// TIA Portal V17 export
// export: Created 2023-05-07T12:12:11.3887996Z, ExportSetting WithDefaults, DisplayName Totally Integrated Automation Portal, DisplayVersion V17, DisplayName TIA Portal Openness, DisplayVersion V17, DisplayName TIA Portal Version Control Interface, DisplayVersion V17, DisplayName TIA Portal Test Suite Advanced, DisplayVersion V17, DisplayName STEP 7 Professional, DisplayVersion V17, DisplayName SIMATIC Energy Suite, DisplayVersion V17, DisplayName STEP 7 Safety, DisplayVersion V17, DisplayName WinCC Professional, DisplayVersion V17
FUNCTION "TrainingFunction" : Void   // FC7, LAD
TITLE = TrainingFunction
{ S7_Optimized_Access := 'TRUE' }
VERSION : 0.1
// stored: AutoNumber true, IsIECCheckEnabled false, SetENOAutomatically false, UDAEnableTagReadback false
BEGIN

REGION Network 1: Call: Training
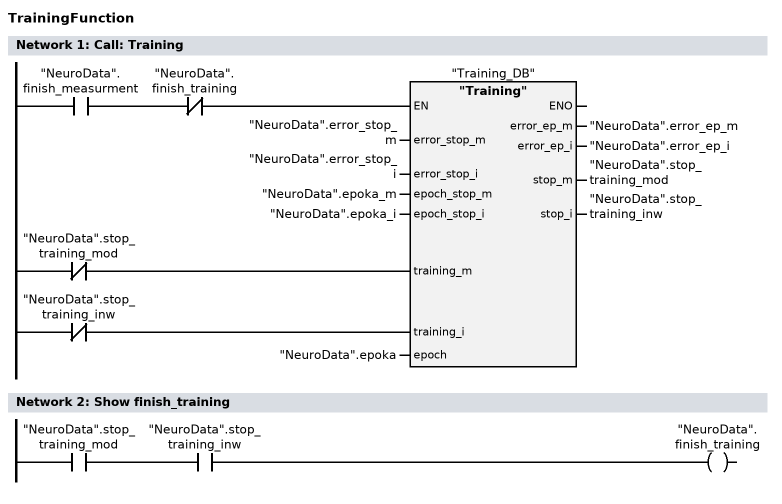
   RUNG wire#powerrail
      Contact( "NeuroData".finish_measurment )
      I_Contact( "NeuroData".finish_training )
      "Training_DB"(training_m := wire#w1, training_i := wire#w2, error_stop_m := "NeuroData".error_stop_m, error_stop_i := "NeuroData".error_stop_i, epoch_stop_m := "NeuroData".epoka_m, epoch_stop_i := "NeuroData".epoka_i, epoch := "NeuroData".epoka, error_ep_m => "NeuroData".error_ep_m, error_ep_i => "NeuroData".error_ep_i, stop_m => "NeuroData".stop_training_mod, stop_i => "NeuroData".stop_training_inw)
   END_RUNG
   RUNG wire#powerrail
      I_Contact( "NeuroData".stop_training_mod )
   END_RUNG wire#w1
   RUNG wire#powerrail
      I_Contact( "NeuroData".stop_training_inw )
   END_RUNG wire#w2
   // the same network as SCL:
   IF "NeuroData".finish_measurment AND NOT "NeuroData".finish_training THEN
       "Training_DB"(error_stop_m := "NeuroData".error_stop_m,   // "Training"
                     error_stop_i := "NeuroData".error_stop_i,
                     epoch_stop_m := "NeuroData".epoka_m,
                     epoch_stop_i := "NeuroData".epoka_i,
                     training_m := NOT "NeuroData".stop_training_mod,
                     training_i := NOT "NeuroData".stop_training_inw,
                     epoch := "NeuroData".epoka,
                     error_ep_m => "NeuroData".error_ep_m,
                     error_ep_i => "NeuroData".error_ep_i,
                     stop_m => "NeuroData".stop_training_mod,
                     stop_i => "NeuroData".stop_training_inw);
   END_IF;
END_REGION

REGION Network 2: Show finish_training
   RUNG wire#powerrail
      Contact( "NeuroData".stop_training_mod )
      Contact( "NeuroData".stop_training_inw )
      Coil( "NeuroData".finish_training )
   END_RUNG
   // the same network as SCL:
   "NeuroData".finish_training := "NeuroData".stop_training_mod AND "NeuroData".stop_training_inw;
END_REGION
END_FUNCTION
